// SIMATIC STEP 7 (V5.x) project T13 E 25
// program: Programa S7(1)

SYMBOL_TABLE
"FLANCOS"	DB 1	DB 1
"MANIOBRA"	DB 2	DB 2
"MEMORIA"	DB 3	DB 3
"MARCHA"	I 0.0	BOOL
"PARO"	I 0.1	BOOL
"DESACTIVACION"	I 0.2	BOOL
"FCEL1"	I 0.3	BOOL
"FCEL2"	I 0.4	BOOL
"FCFLINEA"	I 0.5	BOOL
"SPRESION"	I 0.6	BOOL
"FCT2"	I 0.7	BOOL
"FCT3"	I 1.0	BOOL
"Cycle Execution"	OB 1	OB 1
"CTM1"	Q 0.0	BOOL
"CTM2"	Q 0.1	BOOL
"CTM3"	Q 0.2	BOOL
"PDESPLAZAMIENTO"	Q 0.3	BOOL
"PELEVACION"	Q 0.4	BOOL
"PT2"	Q 0.5	BOOL
"PT3"	Q 0.6	BOOL
END_SYMBOL_TABLE
